// SIMATIC S7-200 project (STEP 7-Micro/WIN), CPU 221 REL 01.10

ORGANIZATION_BLOCK 主程序:OB1
TITLE=程序注释
BEGIN
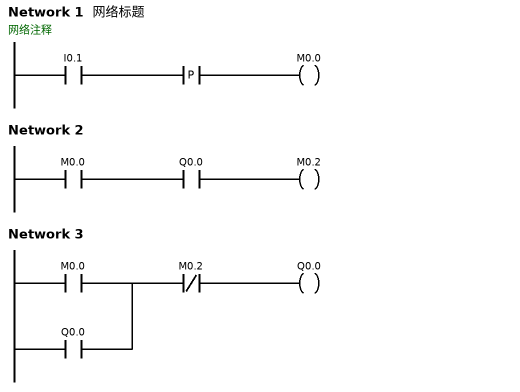
Network 1 // 网络标题
// 网络注释
LD     I0.1
EU
=      M0.0
Network 2
LD     M0.0
A      Q0.0
=      M0.2
Network 3
LD     M0.0
O      Q0.0
AN     M0.2
=      Q0.0
END_ORGANIZATION_BLOCK
